FUNCTION_BLOCK CM_VisionSensor
VAR_INPUT
	SensorInput : DINT;
END_VAR
VAR_OUTPUT
	SensorOutput : DINT;
END_VAR
VAR_IN_OUT
	control_data_vision : CM_Vision_UDT;
END_VAR


SensorOutput := SensorInput;

control_data_vision.PO_PV := SensorOutput;

END_FUNCTION_BLOCK

(* stored: Version 1.1.0.1, ProductVersion 3.1.4024.13
   POU CM_VisionSensor: Id {e05ef0fa-dc49-45cf-a155-8da901e6d7c1}, SpecialFunc None *)
